(* CODESYS project CtaVisHelp_1.0.0.0.library
   DocFormat: reStructuredText
   DefaultNamespace: CtaVisHelp
   Version: 1.0.0.0
   Placeholder: CtaVisHelp
   Company: CTA
   Description: Visu Hilfe Library der CTA
   CompiledLibraryCompatibilityVersion: CODESYS V3.5 SP16 Patch 3
   LanguageModelAttribute: qualified-access-only
   Title: CtaVisHelp
   Author: SIS

Project tree, tasks and I/O mapping:
  libraries: CmpBitmapPool, 3.5.17.0 (System); Visu Utils, 4.5.0.0 (System); Standard, 3.5.18.0 (System); VisuElemBase, * (System); CtaVisSymbols, 1.0.0.0 (CTA); CtaSysConfig, 1.0.0.2 (CTA); VisuSymbols, 4.5.0.0 (System); CtaVisMouseEvent, 1.0.0.0 (CTA)
  40 Visualizations/
    ExklusivParameter/
      visualisation ExkParameterSymbol
    AwakenScreenOnTap/
      BlackScreens/
        visualisation VisSettings
        visualisation VisSmallScreen
        visualisation VisBigScreen
      visualisation PopUpSettings
    Schalter/
      visualisation VIS_DI_Schalter
    BUTTON/
      visualisation VIS_SAFE_BUTTON
  30 Program Organization Units/
    AwakenScreenOnTap/
      function block FB_MOUSINPUT [ST]: HandleMouseBtnEvent, HandleMouseMoveEvent, actConfig, DialogClosed
    BUTTON/
      function block FB_SAFE_BUTTON [ST]: Sichtbar
    CloseDialogue/
      function block FB_CLOSE_DIALOG_ON_MOUSE_OUT [ST]: FB_INIT, HandleMouseBtnEvent, HandleMouseMoveEvent
  00000000-0000-0000-0000-000000000000|D:\CoDeSys\LibrariesV3\trunk\Intern\CAA\CAA Template\3.4.0.0 draft\Placeholder.xml
  00000000-0000-0000-0000-000000000000|D:\CoDeSys\LibrariesV3\trunk\Intern\CAA\CAA Template\3.2.0.3 draft\Prefix.pdf
  00000000-0000-0000-0000-000000000000|D:\CoDeSys\LibrariesV3\trunk\Intern\CAA\CAA Template\3.5.2.0 draft\Placeholder.xml
  20 Structs/
    AwakenScreenOnTap/
      data type scParameter
  50 Images/
  10 Documenation/
    global variables VersionHistory
    global variables readMe
  21 Interface/
  11 Library Parameter/
  12 Konstanten/
  60 Textlisten/
    PRG/
  13 Globale Variablen/
    AwakenScreenOnTap/
      global variables GVL_DarkScreen
    CloseDialogue/
      global variables GVL_DIALOG_CLOSE_ON_MOUSE_EVENT
  5ce3da45-db07-42e7-a21c-a00fff4ed8f6|Icons\alert.svg
  5ce3da45-db07-42e7-a21c-a00fff4ed8f6|Icons\arrow-down.svg
  5ce3da45-db07-42e7-a21c-a00fff4ed8f6|Icons\arrow-down_square.svg
  5ce3da45-db07-42e7-a21c-a00fff4ed8f6|Icons\arrow-left_solo_black.svg
  5ce3da45-db07-42e7-a21c-a00fff4ed8f6|Icons\arrow-right_solo_black.svg
  5ce3da45-db07-42e7-a21c-a00fff4ed8f6|Icons\arrow-up.svg
  5ce3da45-db07-42e7-a21c-a00fff4ed8f6|Icons\calendar-range.svg
  5ce3da45-db07-42e7-a21c-a00fff4ed8f6|Icons\check.svg
  5ce3da45-db07-42e7-a21c-a00fff4ed8f6|Icons\clock-outline.svg
  5ce3da45-db07-42e7-a21c-a00fff4ed8f6|Icons\close_solo_black.svg
  5ce3da45-db07-42e7-a21c-a00fff4ed8f6|Icons\CtaInfo.svg
  5ce3da45-db07-42e7-a21c-a00fff4ed8f6|Icons\database_black.svg
  5ce3da45-db07-42e7-a21c-a00fff4ed8f6|Icons\delete_solo_black.svg
  5ce3da45-db07-42e7-a21c-a00fff4ed8f6|Icons\engine.svg
  5ce3da45-db07-42e7-a21c-a00fff4ed8f6|Icons\front_hand_Black.svg
  5ce3da45-db07-42e7-a21c-a00fff4ed8f6|Icons\front_hand_Yellow_Off.svg
  5ce3da45-db07-42e7-a21c-a00fff4ed8f6|Icons\gear.svg
  5ce3da45-db07-42e7-a21c-a00fff4ed8f6|Icons\home.svg
  5ce3da45-db07-42e7-a21c-a00fff4ed8f6|Icons\information-variant.svg
  5ce3da45-db07-42e7-a21c-a00fff4ed8f6|Icons\lightning-bolt-circle.svg
  5ce3da45-db07-42e7-a21c-a00fff4ed8f6|Icons\message.svg
  5ce3da45-db07-42e7-a21c-a00fff4ed8f6|Icons\message-alert-variant.svg
  5ce3da45-db07-42e7-a21c-a00fff4ed8f6|Icons\minus_solo_black.svg
  5ce3da45-db07-42e7-a21c-a00fff4ed8f6|Icons\plus_solo_black.svg
  5ce3da45-db07-42e7-a21c-a00fff4ed8f6|Icons\power_solo_black.svg
  5ce3da45-db07-42e7-a21c-a00fff4ed8f6|Icons\refresh_solo_black.svg
  5ce3da45-db07-42e7-a21c-a00fff4ed8f6|Icons\SearchFilter.svg
  5ce3da45-db07-42e7-a21c-a00fff4ed8f6|Icons\signal-celular-alt.svg
  5ce3da45-db07-42e7-a21c-a00fff4ed8f6|Icons\toggle-switch.svg
  5ce3da45-db07-42e7-a21c-a00fff4ed8f6|Icons\Modbus_Organization_Logo.svg
  5ce3da45-db07-42e7-a21c-a00fff4ed8f6|Icons\CheckboxUnchecked_withe.svg
  5ce3da45-db07-42e7-a21c-a00fff4ed8f6|Icons\lock_open_black.svg
  5ce3da45-db07-42e7-a21c-a00fff4ed8f6|Icons\check_green.svg
  5ce3da45-db07-42e7-a21c-a00fff4ed8f6|Icons\filter_black.svg
  5ce3da45-db07-42e7-a21c-a00fff4ed8f6|Icons\CtaLogo.png
  5ce3da45-db07-42e7-a21c-a00fff4ed8f6|Icons\Grafana_Logo.svg
  5ce3da45-db07-42e7-a21c-a00fff4ed8f6|Icons\hourglass_top.svg
  text list GlobalTextList
  70_PRG/
    program CalsPRG [ST]
*)

// 20 Structs/AwakenScreenOnTap/scParameter
TYPE scParameter :
	STRUCT
		fbxIsBigScreen			:	CtaSysConfig.fbBOOL;
		fbtBlackScreenDelay		:	CtaSysConfig.fbTIME;
	END_STRUCT
END_TYPE

// 10 Documenation/VersionHistory
(* 

.. image:: ../../Images/CTA_Logo.jpg
   :align: right
   :width: 15% 

**Vorlage**   


============ =========== =========== ============================================
**Date**     **Version** **Author**  **Change**
------------ ----------- ----------- --------------------------------------------
04.03.2021   0.0.0.0     SIS         Vorlage erstellt

============ =========== =========== ============================================


*)
VAR_GLOBAL
    stInfo : STRING:= '0.0.0.0, Vorlage, CTA';
END_VAR

// 10 Documenation/readMe
(*

**ReadMe**
 
|	**Empfehlung**
|
|	Dokumentrieren Sie die Library für eine nachhaltige Entwicklung
|     
| *Beispiel*
| 
| Dies ist die Vorlage Library der CTA. Erstellen Sie ihre Library anhand dieser Vorlage.
*)

VAR_GLOBAL
    xReadMeDone              :   BOOL;
END_VAR

// 13 Globale Variablen/AwakenScreenOnTap/GVL_DarkScreen
{attribute 'qualified_only'}
{attribute 'linkalways'}
VAR_GLOBAL
	fbDarkScreen	:	FB_MOUSINPUT;
END_VAR

// 13 Globale Variablen/CloseDialogue/GVL_DIALOG_CLOSE_ON_MOUSE_EVENT
{attribute 'qualified_only'}
{attribute 'linkalways'}
VAR_GLOBAL
	FB_CLOSE_DIALOG_ON_MOUSE_OUT	:	FB_CLOSE_DIALOG_ON_MOUSE_OUT;
END_VAR

// 30 Program Organization Units/AwakenScreenOnTap/FB_MOUSINPUT
FUNCTION_BLOCK FB_MOUSINPUT EXTENDS CtaVisMouseEvent.FB_MOUSE_EVENT_NODE IMPLEMENTS CtaVisMouseEvent.ITF_MOUSE_EVENT_NODE , VisuElemBase.IDialogCloseListener
VAR
	TON_TIMEOUT		:	Standard.TON;
	xInitDone		:	BOOL;
	xMouseEvent		:	BOOL;
	fbSwitchVisu	:	VU.FbOpenDialogExtended;
	fbConfigFile	:	CtaSysConfig.fbConfigFile;
	scParameter		:	scParameter;
	xIsOpen			:	BOOL;
END_VAR

actConfig();

TON_TIMEOUT(IN := NOT TON_TIMEOUT.Q AND NOT xMouseEvent AND NOT xIsOpen,
			PT := scParameter.fbtBlackScreenDelay.proValue);
			
IF TON_TIMEOUT.Q THEN
	fbSwitchVisu.xExecute := TRUE;
END_IF;

fbSwitchVisu(itfClientFilter := VU.Globals.AllClients,xModal:= FALSE,sDialogName := SEL(scParameter.fbxIsBigScreen.proValue = TRUE,'CtaVisHelp.VisSmallScreen','CtaVisHelp.VisBigScreen'),itfDialogCloseListener := THIS^);

IF fbSwitchVisu.xDone THEN
	fbSwitchVisu.xExecute := FALSE;
	xIsOpen				  := TRUE;
END_IF

xMouseEvent := FALSE;

/// This method will be called when a mouse button is pressed. 
/// RETURN: 
/// TRUE - When the handler has handled this event and it should not be handled by someone else
/// FALSE - When the event is not handled by this handler
METHOD HandleMouseBtnEvent : BOOL
VAR_INPUT
	/// The event type. The value is true if a mouse button was released.
	bMouseUpEvent	: BOOL;
	/// Information about the button that was pressed or released. At the moment this
	/// value is not yet used and will always have the value 0!
	btMouseBtn		: BYTE;
	/// The position where the mouse event was raised. The coordinates of this point are relative to the 
	/// currently active toplevel visualization, even when best fit is activated.  
	ptMouse			: VisuElemBase.VisuStructPoint;
	/// A pointer to the client structure were the event occurred.
	pClient			: POINTER TO VisuElemBase.VisuStructClientData;
	EVENT_TYPE		: CtaVisMouseEvent.enEventType;
END_VAR
IF bMouseUpEvent AND EVENT_TYPE = CtaVisMouseEvent.enEventType.MOUSE_UP THEN
	xMouseEvent := TRUE;
	HandleMouseBtnEvent := FALSE;
END_IF;
END_METHOD

/// This method will be called when the mouse was moved. 
/// RETURN: 
/// TRUE - When the handler has handled this event and it should not be handled by someone else
/// FALSE - When the event is not handled by this handler
METHOD HandleMouseMoveEvent : BOOL
VAR_INPUT
	/// The position where the mouse was moved to. The coordinates of this point are relative to the 
	/// currently active toplevel visualization, even when best fit is activated.  
	ptMouse: VisuElemBase.VisuStructPoint;
	/// A pointer to the client structure were the event occurred.
	pClient: POINTER TO VisuElemBase.VisuStructClientData;
END_VAR
END_METHOD

ACTION actConfig:
fbConfigFile();

scParameter.fbxIsBigScreen		(_usiParaNr := 1,itfConfigFb := fbConfigFile,_WertInit := FALSE);
scParameter.fbtBlackScreenDelay	(_usiParaNr	:= 2,itfConfigFb := fbConfigFile,_WertInit := T#5M);
END_ACTION

(* Notification, that a dialog is closed.*)
METHOD DialogClosed
VAR_INPUT
	(* The IVisualisationDialog instance, that was closed*)
	itfDialog	: VisuElemBase.IVisualisationDialog;
	(* A pointer to the client data*)
	pClientData	: POINTER TO VisuElemBase.VisuStructClientData;
END_VAR
xIsOpen := FALSE;
END_METHOD

END_FUNCTION_BLOCK

// 30 Program Organization Units/BUTTON/FB_SAFE_BUTTON
FUNCTION_BLOCK FB_SAFE_BUTTON
VAR_INPUT
	xSchaltung		:	BOOL;
END_VAR
VAR_OUTPUT
	iState			:	INT;
	xMouseDownTime	:	BOOL;
	xFarbWechsel	:	BOOL;
	dwRamenAus		:	DWORD:= 16#FF000000;
	dwFeldAus		:	DWORD:= 16#FF909191;
	dwRamenEin		:	DWORD:= 16#FF000000;
	dwFeldEin		:	DWORD:= 16#FF80FF80;
	tonBlink		:	Standard.TON;
	tonPress		:	Standard.TON;
	tonTimeOut		:	Standard.TON;
END_VAR
VAR
	usiCase			:	USINT;
END_VAR

METHOD Sichtbar : BOOL
VAR_IN_OUT
	xStateInOut	:	BOOL;
END_VAR
CASE usiCase OF
	0:	// Wait on Input
		tonPress(IN := xSchaltung,	PT := T#1S);
		(* fill bar *)
		IF tonPress.IN THEN
			xMouseDownTime := TRUE;
			iState		   := TO_INT(tonPress.ET);
		END_IF;
		// Resett
		IF NOT xSchaltung AND xMouseDownTime THEN
			usiCase := 4;
		END_IF;
		(* Press done set Color *)
		IF tonPress.Q THEN 
			dwRamenAus 	:= 16#FF000000;	// Black
			dwFeldAus	:= 16#FF909191;	// DarkGray
			dwRamenEin 	:= 16#FF000000;	// Black
			dwFeldEin	:= 16#FF80FFFF;	// Blue					
			usiCase := usiCase + 1;
		END_IF;
		
	1:	// Wait on release and Blink
		(* Blink *)
		tonBlink(	IN	:= NOT tonBlink.Q	,PT := T#500MS);
		(* Schaltung *)
		IF NOT xSchaltung THEN
			usiCase := usiCase + 1;
		END_IF;
	2:	// Wait on second Press
		(* Resett *)
		xMouseDownTime := FALSE;
		(* Blink *)
		tonBlink(	IN	:= NOT tonBlink.Q	,PT := T#500MS);
		(* Timeout *)
		tonTimeOut(	IN 	:= TRUE				, PT := T#20S);
		(* Switch and set Color *)
		IF tonTimeOut.Q OR xSchaltung THEN
			// Schaltung
			IF xSchaltung THEN 
				xStateInOut := NOT xStateInOut;
			END_IF;	
			dwRamenAus 		:= 16#FF000000;	// Black
			dwFeldAus		:= 16#FF909191;	// DarkGray
			dwRamenEin 		:= 16#FF000000;	// Black
			dwFeldEin		:= 16#FF80FF80;	// Green
			usiCase 		:= usiCase + 1;	
		END_IF;

	3:	// Release
		IF NOT xSchaltung THEN
			usiCase := usiCase + 1;
		END_IF;	
	4:	// Resett
		xMouseDownTime 	:= FALSE;
		iState			:= 0;
		tonPress(	IN 	:= FALSE	,PT := T#0S);
		tonBlink(	IN	:= FALSE	,PT := T#0S);
		tonTimeOut(	IN 	:= FALSE	,PT := T#0S);
		IF NOT tonBlink.Q AND NOT tonPress.Q AND NOT tonTimeOut.Q THEN
			usiCase := 0;
		END_IF;
END_CASE

(* Color *)
IF tonBlink.Q THEN
	xFarbWechsel := NOT xFarbWechsel;
ELSIF usiCase = 0 OR usiCase >= 3 THEN
	xFarbWechsel := xStateInOut;
END_IF;
END_METHOD

END_FUNCTION_BLOCK

// 30 Program Organization Units/CloseDialogue/FB_CLOSE_DIALOG_ON_MOUSE_OUT
FUNCTION_BLOCK FB_CLOSE_DIALOG_ON_MOUSE_OUT EXTENDS CtaVisMouseEvent.FB_MOUSE_EVENT_NODE 
VAR_INPUT
END_VAR
VAR_OUTPUT
END_VAR
VAR
	IDialogManager			:	VisuElemBase.IDialogManager10;	
	xAdded					:	BOOL;
END_VAR

//FB_Init ist immer implizit verfügbar und wird primär für die Initialisierung verwendet.
//Der Rückgabewert wird nicht ausgewertet. Für gezielte Einflussnahme können Sie
//die Methoden explizit deklarieren und darin mit dem Standard-Initialisierungscode 
//zusätzlichen Code bereitstellen. Sie können den Rückgabewert auswerten.
METHOD FB_Init: BOOL
VAR_INPUT    
bInitRetains: BOOL; // TRUE: Die Retain-Variablen werden initialisiert (Reset warm / Reset kalt)    
bInCopyCode: BOOL;  // TRUE: Die Instanz wird danach in den Kopiercode kopiert (Online-Change)
END_VAR
VAR
	IDialogManagerTemp : VisuElemBase.IDialogManager;
END_VAR
IDialogManagerTemp :=VisuElemBase.g_VisuManager.GetDialogManager();
__QUERYINTERFACE(IDialogManagerTemp,IDialogManager);
END_METHOD

(* This method will be called when a mouse button is pressed. 
 RETURN: 
 TRUE - When the handler has handled this event and it should not be handled by someone else
 FALSE - When the event is not handled by this handler*)
METHOD HandleMouseBtnEvent : BOOL
VAR_INPUT
	(* The event type. The value is true if a mouse button was released.*)
	bMouseUpEvent	: BOOL;
	(* Information about the button that was pressed or released. At the moment this
 value is not yet used and will always have the value 0!*)
	btMouseBtn		: BYTE;
	(* The position where the mouse event was raised. The coordinates of this point are relative to the 
 currently active toplevel visualization, even when best fit is activated.  *)
	ptMouse			: VisuElemBase.VisuStructPoint;
	(* A pointer to the client structure were the event occurred.*)
	pClient			: POINTER TO VisuElemBase.VisuStructClientData;
	EVENT_TYPE		: CtaVisMouseEvent.enEventType;
END_VAR
VAR
	IDialog			:	VisuElemBase.IvisualisationDialog;
	pRectangle		:	VisuElemBase.VisuStructSimpleRectangle;
	pBottom			:	VisuElemBase.VisuStructPoint;
	pRect			:	VisuElemBase.VisuStructPoint;
	diLow			:	DINT;
	diUp			:	DINT;
	diFor			:	DINT;
END_VAR
IF bMouseUpEvent AND EVENT_TYPE = CtaVisMouseEvent.enEventType.MOUSE_UP THEN
	IF NOT ptMouse.iX.15 AND NOT ptMouse.iY.15 THEN
		IF pClient^.GlobalData.TopMostDialogInfo.InTopMostDialog THEN
			diLow := 0;
			diUp  := pClient^.GlobalData.DialogData.STATIC_NUM_CONCURRENTDIALOGS;
			IF __QUERYINTERFACE(IDialogManager,IDialogManager) THEN
				FOR diFor := diLow TO diUp DO
					IF pClient^.GlobalData.DialogData._staticDialogInfoArray[diFor].info.Dialog = 0 THEN
						EXIT;
					ELSE	
						IF IDialogManager.IsDialogOpen(pClient,pClient^.GlobalData.DialogData._staticDialogInfoArray[diFor].info.Dialog) THEN
							IDialog := pClient^.GlobalData.DialogData._staticDialogInfoArray[diFor].info.Dialog;
							pRect 	:= pClient^.GlobalData.DialogData._staticDialogInfoArray[diFor].info.Rect.ptTopLeft;
						END_IF;
					END_IF;
				END_FOR;
				
				IF __QUERYINTERFACE(IDialog,IDialog) THEN
					pRectangle := IDialog.GetSurroundingRect();
					pBottom    := IDialog.GetSize();
					IF pRect.iX <> 0 OR pRect.iY <> 0 THEN
						IF 	ptMouse.iX < pRect.iX + pRectangle.ptTopLeft.iX		OR
							ptMouse.iY < pRect.iY + pRectangle.ptTopLeft.iY		OR
							ptMouse.iX > pRect.iX + pRectangle.ptBottomRight.iX	OR
							ptMouse.iY > pRect.iY + pRectangle.ptBottomRight.iY	THEN
							IDialogManager.CloseDialog(IDialog,pClient);		
						END_IF;					
					ELSE
						IF 	ptMouse.iX < (pClient^.rClientRect.ptBottomRight.iX - pBottom.iX)/2 + pRectangle.ptTopLeft.iX		OR
							ptMouse.iY < (pClient^.rClientRect.ptBottomRight.iY - pBottom.iY)/2 + pRectangle.ptTopLeft.iY		OR
							ptMouse.iX > (pClient^.rClientRect.ptBottomRight.iX - pBottom.iX)/2 + pRectangle.ptBottomRight.iX	OR
							ptMouse.iY > (pClient^.rClientRect.ptBottomRight.iY - pBottom.iY)/2 + pRectangle.ptBottomRight.iY	THEN
							IDialogManager.CloseDialog(IDialog,pClient);		
						END_IF;
					END_IF;
				END_IF;
			END_IF;
		END_IF;
	END_IF;
END_IF;

HandleMouseBtnEvent := FALSE;
END_METHOD

(* This method will be called when the mouse was moved. 
 RETURN: 
 TRUE - When the handler has handled this event and it should not be handled by someone else
 FALSE - When the event is not handled by this handler*)
METHOD HandleMouseMoveEvent : BOOL
VAR_INPUT
	(* The position where the mouse was moved to. The coordinates of this point are relative to the 
 currently active toplevel visualization, even when best fit is activated.  *)
	ptMouse	: VisuElemBase.VisuStructPoint;
	(* A pointer to the client structure were the event occurred.*)
	pClient	: POINTER TO VisuElemBase.VisuStructClientData;
END_VAR
END_METHOD

END_FUNCTION_BLOCK

// 70_PRG/CalsPRG
PROGRAM CalsPRG
VAR
END_VAR

GVL_DarkScreen.fbDarkScreen();
GVL_DIALOG_CLOSE_ON_MOUSE_EVENT.FB_CLOSE_DIALOG_ON_MOUSE_OUT();

END_PROGRAM

// 40 Visualizations/ExklusivParameter/ExkParameterSymbol
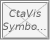
VISUALIZATION ExkParameterSymbol  // 50x40
VAR_INPUT
	stExklParameter		:	STRING[40];
END_VAR
VAR
    fbDialogOpen    		:   VU.FbOpenDialog;
END_VAR
    Image (2,2 46x36), invisible if: stExklParameter = ' ', image: CtaVisSymbols.ImagePool.Settings+
        OnMouseClick: execute {
            fbDialogOpen(	itfClientFilter            	:= VU.Globals.CurrentClient,
                    	 	xExecute                   	:= FALSE,
                    	 	sDialogName                	:= stExklParameter,
            			 	xModal						:= TRUE);
            fbDialogOpen(	itfClientFilter            	:= VU.Globals.CurrentClient,
                     		xExecute                  	:= TRUE,
                     		sDialogName               	:= stExklParameter,
            				xModal						:= TRUE);
        }
END_VISUALIZATION

// 40 Visualizations/AwakenScreenOnTap/BlackScreens/VisSettings
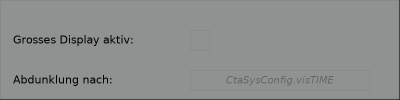
VISUALIZATION VisSettings  // 400x100
VAR_IN_OUT
	fbBlackScreenIn		: 	FB_MOUSINPUT;
END_VAR
    Rectangle (0,0 400x100)
    Label (10,30 150x20), "Grosses Display aktiv:"
    Label (10,70 150x20), "Abdunklung nach:"
    Frame (190,30 20x20)
        shows CtaSysConfig.visBOOL(visfbBOOLIn := fbBlackScreenIn.scParameter.fbxIsBigScreen)
    Frame (190,70 180x20)
        shows CtaSysConfig.visTIME(visfbTIMEIn := fbBlackScreenIn.scParameter.fbtBlackScreenDelay)
END_VISUALIZATION

// 40 Visualizations/AwakenScreenOnTap/BlackScreens/VisSmallScreen
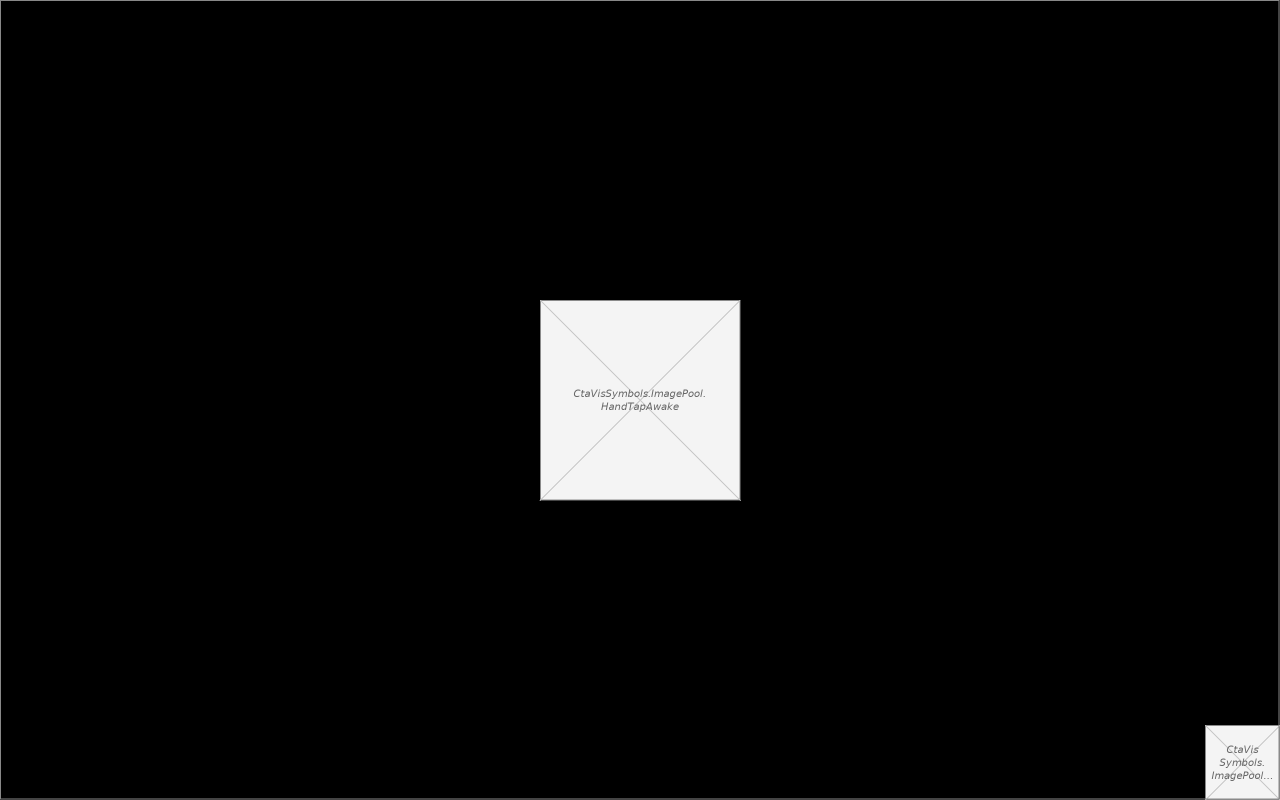
VISUALIZATION VisSmallScreen  // 1280x800
    Rectangle (0,0 1280x800)
        OnMouseDown:  Dialog=Current Dialog, Result=OK, NumpadKeypadSet=True
    Image (540,300 200x200), image: CtaVisSymbols.ImagePool.HandTapAwake
        OnMouseDown:  Dialog=Current Dialog, Result=OK, NumpadKeypadSet=True
    Image (1205,725 75x75), image: CtaVisSymbols.ImagePool.gear_white
        OnMouseDown:  Dialog=PopUpSettings, OpenModal=True, OpenCentered=True
END_VISUALIZATION

// 40 Visualizations/AwakenScreenOnTap/BlackScreens/VisBigScreen
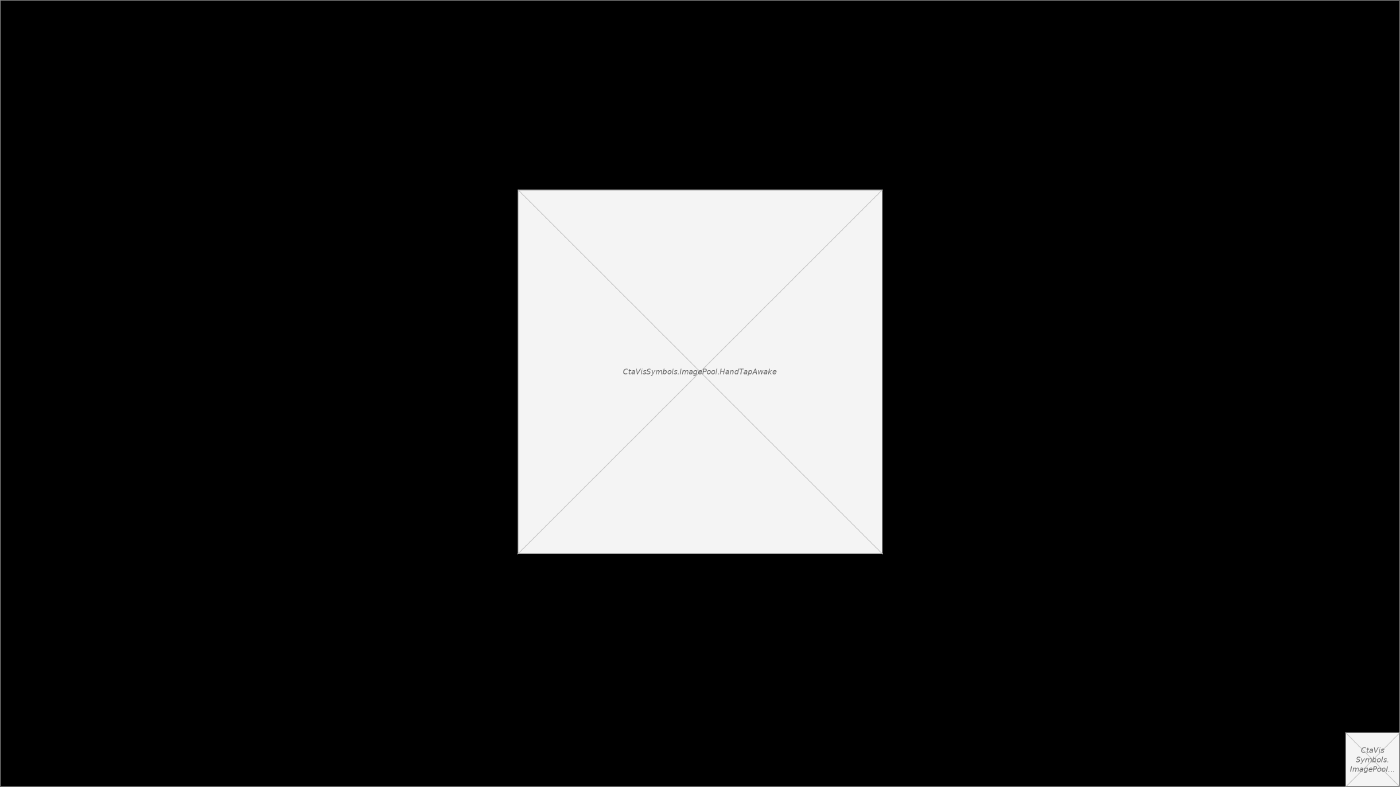
VISUALIZATION VisBigScreen  // 1920x1080
    Rectangle (0,0 1920x1080)
        OnMouseDown:  Dialog=Current Dialog, Result=OK, NumpadKeypadSet=True
    Image (710,260 500x500), image: CtaVisSymbols.ImagePool.HandTapAwake
        OnMouseDown:  Dialog=Current Dialog, Result=OK, NumpadKeypadSet=True
    Image (1845,1005 75x75), image: CtaVisSymbols.ImagePool.gear_white
        OnMouseDown:  Dialog=PopUpSettings, OpenModal=True, OpenCentered=True
END_VISUALIZATION

// 40 Visualizations/AwakenScreenOnTap/PopUpSettings
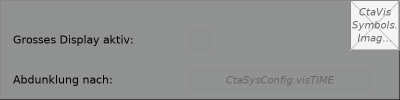
VISUALIZATION PopUpSettings  // 400x100
    Frame (0,0 400x100)
        shows VisSettings(fbBlackScreenIn := GVL_DarkScreen.fbDarkScreen)
    Image (350,0 50x50), image: CtaVisSymbols.ImagePool.close_solo_black
        OnMouseDown:  Dialog=Current Dialog, Result=OK, NumpadKeypadSet=True
END_VISUALIZATION

// 40 Visualizations/Schalter/VIS_DI_Schalter
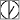
VISUALIZATION VIS_DI_Schalter  // 20x20
VAR_INPUT
	xDI		:	BOOL;	
END_VAR
    Ellipse (0,0 19x19), colour toggle: xDI
    Line (9,6) (9,0)
    Line (9,19) (9,14)
    Line (9,14) (14,6), invisible if: xDI
    Line (9,14) (9,6), invisible if: NOT xDI
END_VISUALIZATION

// 40 Visualizations/BUTTON/VIS_SAFE_BUTTON
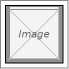
VISUALIZATION VIS_SAFE_BUTTON  // 69x69
VAR_INPUT CONSTANT
	stImage			: STRING := 'CtaVisSymbols.ImagePool.power_solo_black';
END_VAR
VAR_IN_OUT
	xState			: BOOL;
END_VAR
VAR
	fbButton		: FB_SAFE_BUTTON;
END_VAR
    RoundedRectangle (0,0 68x68)
    RoundedRectangle (5,5 58x58), colour toggle: fbButton.xFarbWechsel, invisible if: fbButton.Sichtbar(xState), colour variable: fbButton.dwFeldAus
        p3450524324: fbButton.dwRamenAus
        p3092690914: fbButton.dwRamenEin
        p2167032090: fbButton.dwFeldEin
        tap fbButton.xSchaltung
    Progressbar (9,6 50x7), variable: fbButton.iState, invisible if: NOT fbButton.xMouseDownTime
    Image (9,9 50x50)
        p84334746: stImage
        OnMouseLeave: execute { fbButton.xSchaltung := FALSE; }
        OnMouseDown: execute { fbButton.xSchaltung := TRUE; }
        OnMouseUp: execute { fbButton.xSchaltung := FALSE; }
END_VISUALIZATION
